{attribute 'GeneratedUsingTerminal: EL9260-0000-0016'}
{attribute addProperty BoxType "EL9260-0000-0016"}
{attribute addProperty Id "EtcSlaveTerminalBasePowerOKAT %I*PowerOK_CEB2FD121FuseErrorAT %I*FuseError_1EC650DA1WcStateAT %I*WcState_9091E0EB2InfoDataAT %I*InfoData_6F19DB2B2"}
{attribute addProperty CRC "558825041"}
{attribute addProperty Size "6"}
TYPE EL9260_214EFE51 EXTENDS EtcSlaveTerminalBase :
STRUCT
	{attribute addProperty Name "PowerOK"}
	PowerOK : PowerOK_CEB2FD12;
	{attribute addProperty Name "FuseError"}
	FuseError : FuseError_1EC650DA;
	{attribute addProperty Name "WcState"}
	WcState : WcState_9091E0EB;
	{attribute addProperty Name "InfoData"}
	InfoData : InfoData_6F19DB2B;
END_STRUCT
END_TYPE

(* stored: Version 1.2.0.0, ProductVersion 3.1.4024.9
   DUT EL9260_214EFE51: Id {750cd5a1-9c22-4265-b047-e855c0ea10d6} *)
